(* IEC 61131-3 sources: InfiniteStateMachine/extracted_st/project/library_information, 1 file *)

(* ---- getlibversion-GetLibVersion.st ---- *)
(* --- Interface --- *)
// This function has been automatically generated from the project information.
FUNCTION GetLibVersion : VERSION
VAR_INPUT

END_VAR

(* --- Implementation --- *)
GetLibVersion.uiMajor := 0;
GetLibVersion.uiMinor := 1;
GetLibVersion.uiServicePack := 1;
GetLibVersion.uiPatch := 1;
